{attribute addProperty BoxType "EL6201-0000-0017"}
{attribute addProperty Id "Slave_3A_DI0BIT10.12517Slave_3A_DI1BIT10.12518Slave_3A_DI2BIT10.12519Slave_3A_DI3BIT10.12520Slave_3B_DI0BIT10.12521Slave_3B_DI1BIT10.12522Slave_3B_DI2BIT10.12523Slave_3B_DI3BIT10.12524"}
{attribute addProperty CRC "166721144"}
{attribute addProperty SizeInBites "8"}
{attribute addProperty SizeInBytes "1"}
TYPE Slave_3_Inputs_09EFF678 :
STRUCT
	{attribute addProperty Name "Slave_3A_DI0"}
	Slave_3A_DI0 : BIT;
	{attribute addProperty Name "Slave_3A_DI1"}
	Slave_3A_DI1 : BIT;
	{attribute addProperty Name "Slave_3A_DI2"}
	Slave_3A_DI2 : BIT;
	{attribute addProperty Name "Slave_3A_DI3"}
	Slave_3A_DI3 : BIT;
	{attribute addProperty Name "Slave_3B_DI0"}
	Slave_3B_DI0 : BIT;
	{attribute addProperty Name "Slave_3B_DI1"}
	Slave_3B_DI1 : BIT;
	{attribute addProperty Name "Slave_3B_DI2"}
	Slave_3B_DI2 : BIT;
	{attribute addProperty Name "Slave_3B_DI3"}
	Slave_3B_DI3 : BIT;
END_STRUCT
END_TYPE

(* stored: Version 1.2.0.0, ProductVersion 3.1.4024.9
   DUT Slave_3_Inputs_09EFF678: Id {f2491c5b-4b4a-43f8-a2c3-79bddfa83051} *)
